// TIA Portal V20 export
DATA_BLOCK "InstCallProcessCount"   // DB24
// stored: InstanceOfName CallProcessCount, InstanceOfType FB
"CallProcessCount"
   // VAR
   //    statPulse { ExternalAccessible := 'False'; ExternalVisible := 'False'; ExternalWritable := 'False'} : Array[0..299] of Bool;
   // END_VAR
BEGIN
END_DATA_BLOCK
